% RSLogix 500 project I2P Hands-On 3 - Mitch.RSS, saved by version 10.00.00.00 %
PROJECT "ML01B"    % processor: Bul.1763 MicroLogix 1100 Series B %

PROGRAM FILES
  LAD 2   11 rungs

DATA FILES
  O0 OUTPUT  4 elements
  I1 INPUT  6 elements
  S2 STATUS  66 elements
  B3 BINARY  1 elements
  T4 TIMER  1 elements
  C5 COUNTER  1 elements
  R6 CONTROL  1 elements
  N7 INTEGER  1 elements
  F8 FLOAT  1 elements

LADDER 2
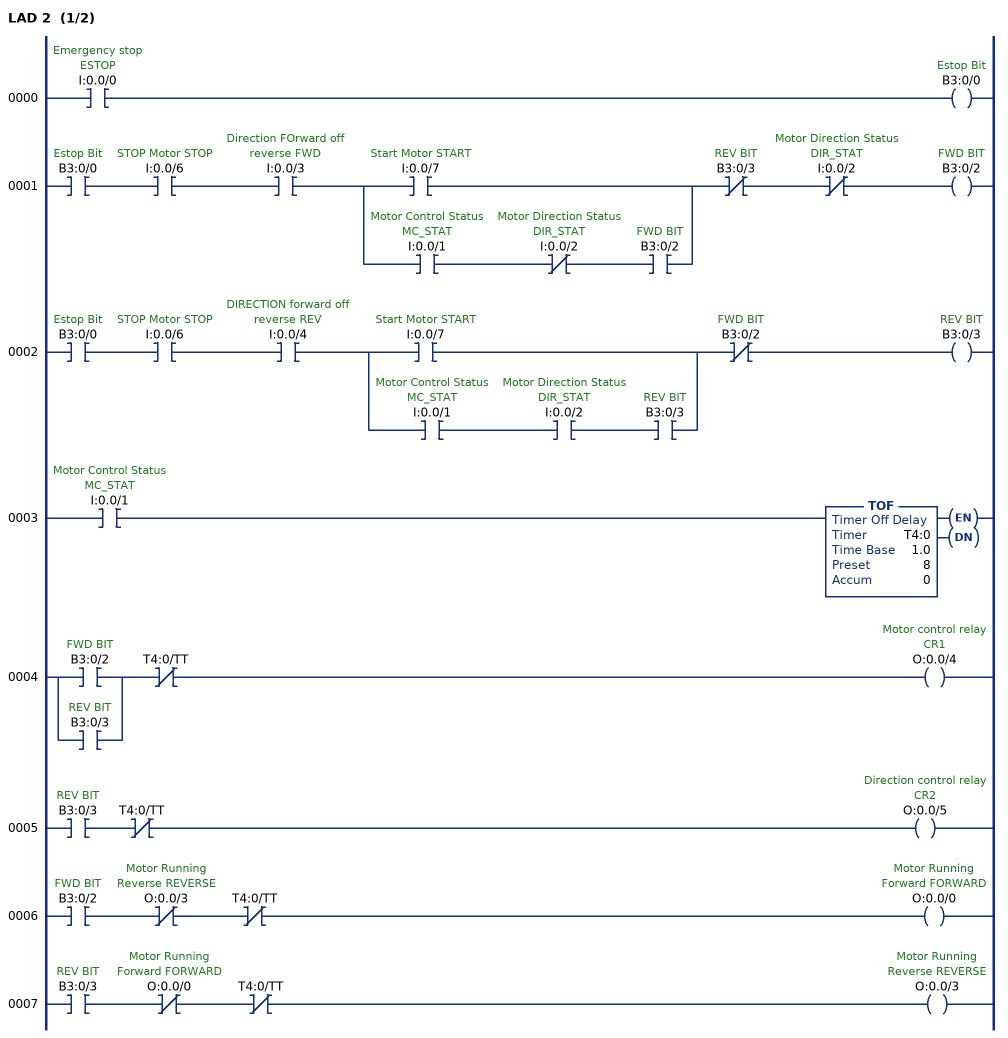
% Rung: 0 %
SOR XIC I:0.0/0 OTE B3:0/0 EOR
%   I:0.0/0  ESTOP  "Emergency stop" %
%   B3:0/0  "Estop Bit" %
% Rung: 1 %
SOR XIC B3:0/0 XIC I:0.0/6 XIC I:0.0/3 BST XIC I:0.0/7 NXB XIC I:0.0/1 XIO I:0.0/2 XIC B3:0/2 BND XIO B3:0/3 XIO I:0.0/2 OTE B3:0/2 EOR
%   B3:0/0  "Estop Bit" %
%   I:0.0/6  STOP  "STOP Motor" %
%   I:0.0/3  FWD  "Direction FOrward off reverse" %
%   I:0.0/7  START  "Start Motor" %
%   I:0.0/1  MC_STAT  "Motor Control Status" %
%   I:0.0/2  DIR_STAT  "Motor Direction Status" %
%   B3:0/2  "FWD BIT" %
%   B3:0/3  "REV BIT" %
% Rung: 2 %
SOR XIC B3:0/0 XIC I:0.0/6 XIC I:0.0/4 BST XIC I:0.0/7 NXB XIC I:0.0/1 XIC I:0.0/2 XIC B3:0/3 BND XIO B3:0/2 OTE B3:0/3 EOR
%   B3:0/0  "Estop Bit" %
%   I:0.0/6  STOP  "STOP Motor" %
%   I:0.0/4  REV  "DIRECTION forward off reverse" %
%   I:0.0/7  START  "Start Motor" %
%   I:0.0/1  MC_STAT  "Motor Control Status" %
%   I:0.0/2  DIR_STAT  "Motor Direction Status" %
%   B3:0/3  "REV BIT" %
%   B3:0/2  "FWD BIT" %
% Rung: 3 %
SOR XIC I:0.0/1 TOF T4:0 1.0 8 0 EOR
%   I:0.0/1  MC_STAT  "Motor Control Status" %
% Rung: 4 %
SOR BST XIC B3:0/2 NXB XIC B3:0/3 BND XIO T4:0/TT OTE O:0.0/4 EOR
%   B3:0/2  "FWD BIT" %
%   B3:0/3  "REV BIT" %
%   O:0.0/4  CR1  "Motor control relay" %
% Rung: 5 %
SOR XIC B3:0/3 XIO T4:0/TT OTE O:0.0/5 EOR
%   B3:0/3  "REV BIT" %
%   O:0.0/5  CR2  "Direction control relay" %
% Rung: 6 %
SOR XIC B3:0/2 XIO O:0.0/3 XIO T4:0/TT OTE O:0.0/0 EOR
%   B3:0/2  "FWD BIT" %
%   O:0.0/3  REVERSE  "Motor Running Reverse" %
%   O:0.0/0  FORWARD  "Motor Running Forward" %
% Rung: 7 %
SOR XIC B3:0/3 XIO O:0.0/0 XIO T4:0/TT OTE O:0.0/3 EOR
%   B3:0/3  "REV BIT" %
%   O:0.0/0  FORWARD  "Motor Running Forward" %
%   O:0.0/3  REVERSE  "Motor Running Reverse" %

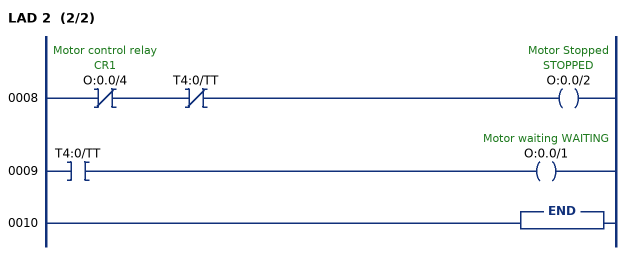
% Rung: 8 %
SOR XIO O:0.0/4 XIO T4:0/TT OTE O:0.0/2 EOR
%   O:0.0/4  CR1  "Motor control relay" %
%   O:0.0/2  STOPPED  "Motor Stopped" %
% Rung: 9 %
SOR XIC T4:0/TT OTE O:0.0/1 EOR
%   O:0.0/1  WAITING  "Motor waiting" %
% Rung: 10 %
SOR END EOR

DATA TABLE (non-zero values as saved)
DATA B3
% B3:0 % 0X0001
DATA T4
% .PRE .ACC %
% T4:0 % 8 0
